FUNCTION_BLOCK FbTxS7con1 //Данные отправленные через S7 connection в NetPro.
TITLE   = 'Данные отправленные через S7 connection в NetPro.'

{//Атрибуты для PCS7.
S7_read_back := 'true' ; //CFC: Chart>Readback активен для прототипов DB.
S7_blockview := 'big'    //CFC: отображение блока маленькое или большое.
}

//Атрибуты для STEP7.
VERSION : '2.1'
AUTHOR  : VA
FAMILY  : LIB_PLC

VAR_INPUT //Входные переменные, сохраняемые.
TX1  :INT := 0; //Отправить значение N1 в удаленный ПЛК.
TX2  :INT := 0; //Отправить значение N2 в удаленный ПЛК.
TX3  :INT := 0; //Отправить значение N3 в удаленный ПЛК.
TX4  :INT := 0; //Отправить значение N4 в удаленный ПЛК.
TX5  :INT := 0; //Отправить значение N5 в удаленный ПЛК.
TX6  :INT := 0; //Отправить значение N6 в удаленный ПЛК.
TX7  :INT := 0; //Отправить значение N7 в удаленный ПЛК.
TX8  :INT := 0; //Отправить значение N8 в удаленный ПЛК.
TX9  :INT := 0; //Отправить значение N9 в удаленный ПЛК.
TX10 :INT := 0; //Отправить значение N10 в удаленный ПЛК.
TX11 :INT := 0; //Отправить значение N11 в удаленный ПЛК.
TX12 :INT := 0; //Отправить значение N12 в удаленный ПЛК.
TX13 :INT := 0; //Отправить значение N13 в удаленный ПЛК.
TX14 :INT := 0; //Отправить значение N14 в удаленный ПЛК.
TX15 :INT := 0; //Отправить значение N15 в удаленный ПЛК.
TX16 :INT := 0; //Отправить значение N16 в удаленный ПЛК.
TX17 :INT := 0; //Отправить значение N17 в удаленный ПЛК.
TX18 :INT := 0; //Отправить значение N18 в удаленный ПЛК.
TX19 :INT := 0; //Отправить значение N19 в удаленный ПЛК.
TX20 :INT := 0; //Отправить значение N20 в удаленный ПЛК.
TX21 :INT := 0; //Отправить значение N21 в удаленный ПЛК.
TX22 :INT := 0; //Отправить значение N22 в удаленный ПЛК.
TX23 :INT := 0; //Отправить значение N23 в удаленный ПЛК.
TX24 :INT := 0; //Отправить значение N24 в удаленный ПЛК.
TX25 :INT := 0; //Отправить значение N25 в удаленный ПЛК.
TX26 :INT := 0; //Отправить значение N26 в удаленный ПЛК.
TX27 :INT := 0; //Отправить значение N27 в удаленный ПЛК.
TX28 :INT := 0; //Отправить значение N28 в удаленный ПЛК.
TX29 :INT := 0; //Отправить значение N29 в удаленный ПЛК.
TX30 :INT := 0; //Отправить значение N30 в удаленный ПЛК.
TX31 :INT := 0; //Отправить значение N31 в удаленный ПЛК.
TX32 :INT := 0; //Отправить значение N32 в удаленный ПЛК.
END_VAR

VAR_OUTPUT //Выходные переменные, сохраняемые.
END_VAR

//Три блока работают совместно.
//FbTxS7con1 FbS7Con1 FbRxS7con1
;

END_FUNCTION_BLOCK

//  +---------+
//  | GNU GPL |
//  +---------+
//  |
//  |
//  .= .-_-. =.
// ((_/)o o(\_))
//  `-'(. .)`-'
//  |/| \_/ |\
//  ( |     | )
//  /"\_____/"\
//  \__)   (__/
// @COPYLEFT ALL WRONGS RESERVED :)
// Author: VA
// Contacts: DIY.PLC.314@gmail.com
// License: GNU GPL v2
//
// https://www.youtube.com/@DIY_PLC
// https://github.com/DIYPLC

